// TIA Portal project "PROGRAMA_P1" (V16)

(* hardware
DEVICE "S7-1200 station_1"  S7-1200 Station
   slot 0: "Rack_0"  S7-1200 Rack  Rack  V1.0
   slot 1: "PLC_1"  CPU 1215C DC/DC/DC  6ES7 215-1AG40-0XB0  V4.4
DEVICE "PC-System_1"  SIMATIC PC station
   slot 0: "Estación PC SIMATIC"  Rail  SIMATIC PC-Station  V1.0
      slot 125: "Stationmanager"  Station_Manager  V6.0.4
   slot 1: "HMI_RT_1"  WinCC RT Advanced  6AV2 104-0xxxx-xxxx  16.0.0.0
      slot 33792: "Interfaz del equipo"  Host interface
   slot 2: "IE general_1"  IE General  IE_CP  V8.2.0
*)

// ===== PLC "PLC_1"  CPU 1215C DC/DC/DC =====

VAR_GLOBAL   // PLC tag table "Tabla de variables estándar"
   "Guardamotor 1Q1" AT %I0.0 : Bool;
   "Detector 1B1" AT %I0.1 : Bool;
   "Detector 1B2" AT %I0.2 : Bool;
   "Fotocelula 1B3" AT %I0.3 : Bool;
   "Pulsador Reinicio 1S1" AT %I0.4 : Bool;
   "Pulsador Paro 1S2" AT %I0.5 : Bool;
   "Contactor Apertura 1KM1" AT %Q0.0 : Bool;
   "Contactor Cerrado 1KM2" AT %Q0.1 : Bool;
   "Piloto 1H1" AT %Q0.2 : Bool;
   "Etapa 0" AT %M10.0 : Bool;
   "Etapa 1" AT %M10.1 : Bool;
   "Etapa 2" AT %M10.2 : Bool;
   "Etapa 3" AT %M10.3 : Bool;
   "Etapa 4" AT %M10.4 : Bool;
   "Etapa 5" AT %M10.5 : Bool;
   "Etapa 6" AT %M10.6 : Bool;
   "Etapa 7" AT %M10.7 : Bool;
   "Etapa 8" AT %M11.0 : Bool;
   "Etapa 9" AT %M11.1 : Bool;
   "Etapa 10" AT %M11.2 : Bool;
   "Etapa 11" AT %M11.3 : Bool;
   "Etapa 12" AT %M11.4 : Bool;
   "Etapa 20" AT %M11.5 : Bool;
   "Etapa 21" AT %M11.6 : Bool;
   "Etapa 22" AT %M11.7 : Bool;
   "System_Byte" AT %MB1 : Byte;
   "FirstScan" AT %M1.0 : Bool;
   "DiagStatusUpdate" AT %M1.1 : Bool;
   "AlwaysTRUE" AT %M1.2 : Bool;
   "AlwaysFALSE" AT %M1.3 : Bool;
   "Clock_Byte" AT %MB0 : Byte;
   "Clock_10Hz" AT %M0.0 : Bool;
   "Clock_5Hz" AT %M0.1 : Bool;
   "Clock_2.5Hz" AT %M0.2 : Bool;
   "Clock_2Hz" AT %M0.3 : Bool;
   "Clock_1.25Hz" AT %M0.4 : Bool;
   "Clock_1Hz" AT %M0.5 : Bool;
   "Clock_0.625Hz" AT %M0.6 : Bool;
   "Clock_0.5Hz" AT %M0.7 : Bool;
   "MB10" AT %MB10 : Byte;
   "MB11" AT %MB11 : Byte;
END_VAR

DATA_BLOCK "Variables"   // DB1
{ S7_Optimized_Access := 'TRUE' }
VERSION : 0.1
   VAR
      MAN : Bool;
      T2Time : Time;
      ActualTime : DTL;
      TimeError : Word;
      Abrir_Manual : Bool;
      Cerrar_Manual : Bool;
      InTime : Bool;
      Flanco_Paro : Bool;
      LeftTime : Time;
   END_VAR
BEGIN
END_DATA_BLOCK

// folder: System blocks/Program resources

DATA_BLOCK "T1"   // DB2
{ S7_Optimized_Access := 'TRUE' }
AUTHOR : Simatic
FAMILY : IEC
NAME : IEC_TMR
VERSION : 1.0
// stored: InstanceOfName IEC_TIMER
"IEC_TIMER"
BEGIN
END_DATA_BLOCK

DATA_BLOCK "T2"   // DB3
{ S7_Optimized_Access := 'TRUE' }
AUTHOR : Simatic
FAMILY : IEC
NAME : IEC_TMR
VERSION : 1.0
// stored: InstanceOfName IEC_TIMER
"IEC_TIMER"
BEGIN
END_DATA_BLOCK

// folder: (top level)

ORGANIZATION_BLOCK "Main"   // OB1, LAD, ProgramCycle
TITLE = "Main Program Sweep (Cycle)"
{ S7_Optimized_Access := 'TRUE' }
VERSION : 0.1
   VAR_INPUT
      Initial_Call : Bool;   // Initial call of this OB
      Remanence : Bool;   // =True, if remanent data are available
   END_VAR
BEGIN

REGION Network 1: SR Etapa 0
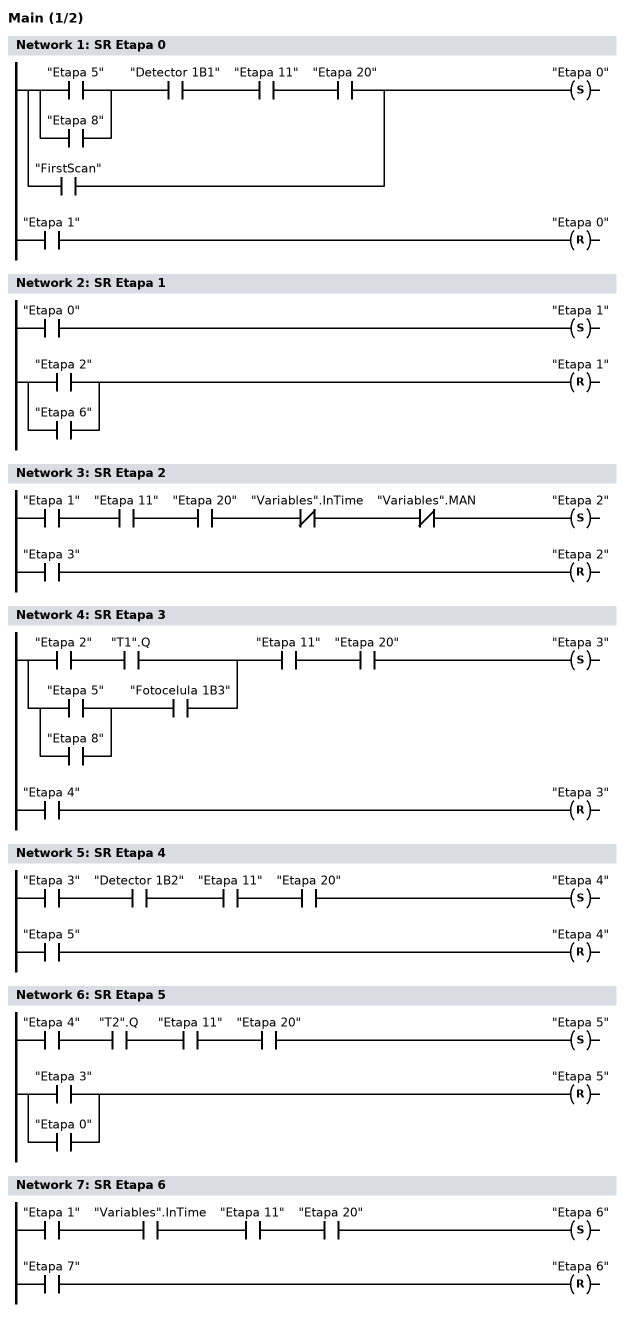
   RUNG wire#powerrail
      Contact( "Etapa 5" )
      wire#w1
      Contact( "Detector 1B1" )
      Contact( "Etapa 11" )
      Contact( "Etapa 20" )
      wire#w2
      S_Coil( "Etapa 0" )
   END_RUNG
   RUNG wire#powerrail
      Contact( "Etapa 8" )
   END_RUNG wire#w1
   RUNG wire#powerrail
      Contact( "FirstScan" )
   END_RUNG wire#w2
   RUNG wire#powerrail
      Contact( "Etapa 1" )
      R_Coil( "Etapa 0" )
   END_RUNG
   // the same network as SCL:
   IF (("Etapa 5" OR "Etapa 8") AND "Detector 1B1" AND "Etapa 11" AND "Etapa 20") OR "FirstScan" THEN
       "Etapa 0" := TRUE;
   END_IF;
   IF "Etapa 1" THEN "Etapa 0" := FALSE; END_IF;
END_REGION

REGION Network 2: SR Etapa 1
   RUNG wire#powerrail
      Contact( "Etapa 0" )
      S_Coil( "Etapa 1" )
   END_RUNG
   RUNG wire#powerrail
      Contact( "Etapa 2" )
      wire#w1
      R_Coil( "Etapa 1" )
   END_RUNG
   RUNG wire#powerrail
      Contact( "Etapa 6" )
   END_RUNG wire#w1
   // the same network as SCL:
   IF "Etapa 0" THEN "Etapa 1" := TRUE; END_IF;
   IF "Etapa 2" OR "Etapa 6" THEN "Etapa 1" := FALSE; END_IF;
END_REGION

REGION Network 3: SR Etapa 2
   RUNG wire#powerrail
      Contact( "Etapa 1" )
      Contact( "Etapa 11" )
      Contact( "Etapa 20" )
      I_Contact( "Variables".InTime )
      I_Contact( "Variables".MAN )
      S_Coil( "Etapa 2" )
   END_RUNG
   RUNG wire#powerrail
      Contact( "Etapa 3" )
      R_Coil( "Etapa 2" )
   END_RUNG
   // the same network as SCL:
   IF "Etapa 1" AND "Etapa 11" AND "Etapa 20" AND NOT "Variables".InTime AND NOT "Variables".MAN THEN
       "Etapa 2" := TRUE;
   END_IF;
   IF "Etapa 3" THEN "Etapa 2" := FALSE; END_IF;
END_REGION

REGION Network 4: SR Etapa 3
   RUNG wire#powerrail
      Contact( "Etapa 2" )
      Contact( "T1".Q )
      wire#w1
      Contact( "Etapa 11" )
      Contact( "Etapa 20" )
      S_Coil( "Etapa 3" )
   END_RUNG
   RUNG wire#powerrail
      Contact( "Etapa 5" )
      wire#w2
      Contact( "Fotocelula 1B3" )
   END_RUNG wire#w1
   RUNG wire#powerrail
      Contact( "Etapa 8" )
   END_RUNG wire#w2
   RUNG wire#powerrail
      Contact( "Etapa 4" )
      R_Coil( "Etapa 3" )
   END_RUNG
   // the same network as SCL:
   IF (("Etapa 2" AND "T1".Q) OR (("Etapa 5" OR "Etapa 8") AND "Fotocelula 1B3")) AND "Etapa 11" AND "Etapa 20" THEN
       "Etapa 3" := TRUE;
   END_IF;
   IF "Etapa 4" THEN "Etapa 3" := FALSE; END_IF;
END_REGION

REGION Network 5: SR Etapa 4
   RUNG wire#powerrail
      Contact( "Etapa 3" )
      Contact( "Detector 1B2" )
      Contact( "Etapa 11" )
      Contact( "Etapa 20" )
      S_Coil( "Etapa 4" )
   END_RUNG
   RUNG wire#powerrail
      Contact( "Etapa 5" )
      R_Coil( "Etapa 4" )
   END_RUNG
   // the same network as SCL:
   IF "Etapa 3" AND "Detector 1B2" AND "Etapa 11" AND "Etapa 20" THEN "Etapa 4" := TRUE; END_IF;
   IF "Etapa 5" THEN "Etapa 4" := FALSE; END_IF;
END_REGION

REGION Network 6: SR Etapa 5
   RUNG wire#powerrail
      Contact( "Etapa 4" )
      Contact( "T2".Q )
      Contact( "Etapa 11" )
      Contact( "Etapa 20" )
      S_Coil( "Etapa 5" )
   END_RUNG
   RUNG wire#powerrail
      Contact( "Etapa 3" )
      wire#w1
      R_Coil( "Etapa 5" )
   END_RUNG
   RUNG wire#powerrail
      Contact( "Etapa 0" )
   END_RUNG wire#w1
   // the same network as SCL:
   IF "Etapa 4" AND "T2".Q AND "Etapa 11" AND "Etapa 20" THEN "Etapa 5" := TRUE; END_IF;
   IF "Etapa 3" OR "Etapa 0" THEN "Etapa 5" := FALSE; END_IF;
END_REGION

REGION Network 7: SR Etapa 6
   RUNG wire#powerrail
      Contact( "Etapa 1" )
      Contact( "Variables".InTime )
      Contact( "Etapa 11" )
      Contact( "Etapa 20" )
      S_Coil( "Etapa 6" )
   END_RUNG
   RUNG wire#powerrail
      Contact( "Etapa 7" )
      R_Coil( "Etapa 6" )
   END_RUNG
   // the same network as SCL:
   IF "Etapa 1" AND "Variables".InTime AND "Etapa 11" AND "Etapa 20" THEN "Etapa 6" := TRUE; END_IF;
   IF "Etapa 7" THEN "Etapa 6" := FALSE; END_IF;
END_REGION

REGION Network 8: SR Etapa 7
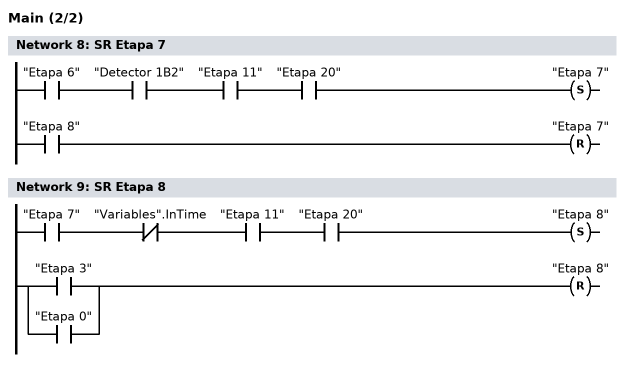
   RUNG wire#powerrail
      Contact( "Etapa 6" )
      Contact( "Detector 1B2" )
      Contact( "Etapa 11" )
      Contact( "Etapa 20" )
      S_Coil( "Etapa 7" )
   END_RUNG
   RUNG wire#powerrail
      Contact( "Etapa 8" )
      R_Coil( "Etapa 7" )
   END_RUNG
   // the same network as SCL:
   IF "Etapa 6" AND "Detector 1B2" AND "Etapa 11" AND "Etapa 20" THEN "Etapa 7" := TRUE; END_IF;
   IF "Etapa 8" THEN "Etapa 7" := FALSE; END_IF;
END_REGION

REGION Network 9: SR Etapa 8
   RUNG wire#powerrail
      Contact( "Etapa 7" )
      I_Contact( "Variables".InTime )
      Contact( "Etapa 11" )
      Contact( "Etapa 20" )
      S_Coil( "Etapa 8" )
   END_RUNG
   RUNG wire#powerrail
      Contact( "Etapa 3" )
      wire#w1
      R_Coil( "Etapa 8" )
   END_RUNG
   RUNG wire#powerrail
      Contact( "Etapa 0" )
   END_RUNG wire#w1
   // the same network as SCL:
   IF "Etapa 7" AND NOT "Variables".InTime AND "Etapa 11" AND "Etapa 20" THEN "Etapa 8" := TRUE; END_IF;
   IF "Etapa 3" OR "Etapa 0" THEN "Etapa 8" := FALSE; END_IF;
END_REGION
END_ORGANIZATION_BLOCK

ORGANIZATION_BLOCK "Temporizadores"   // OB123, LAD, ProgramCycle
TITLE = "Main Program Sweep (Cycle)"
{ S7_Optimized_Access := 'TRUE' }
VERSION : 0.1
   VAR_INPUT
      Initial_Call : Bool;   // Initial call of this OB
      Remanence : Bool;   // =True, if remanent data are available
   END_VAR
BEGIN

REGION Network 1: Temporizador 1
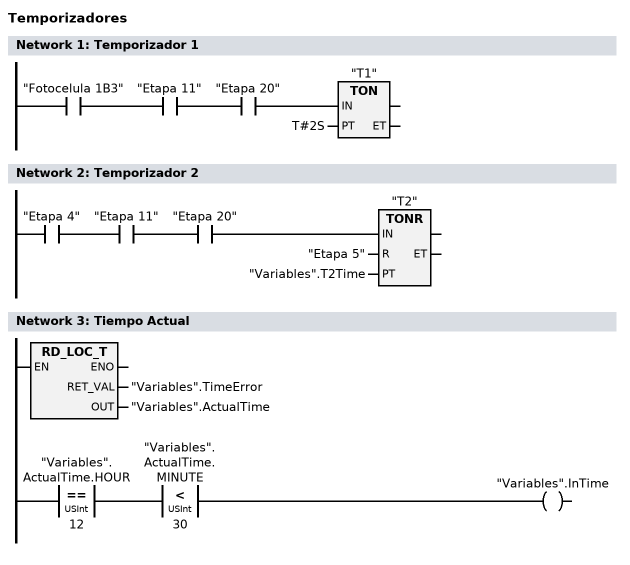
   "T1".TON(IN := "Fotocelula 1B3" AND "Etapa 11" AND "Etapa 20", PT := T#2S);
END_REGION

REGION Network 2: Temporizador 2
   "T2".TONR(IN := "Etapa 4" AND "Etapa 11" AND "Etapa 20", R := "Etapa 5", PT := "Variables".T2Time);
END_REGION

REGION Network 3: Tiempo Actual
   "Variables".TimeError := RD_LOC_T(OUT => "Variables".ActualTime);
   "Variables".InTime := ("Variables".ActualTime.HOUR = 12) AND ("Variables".ActualTime.MINUTE < 30);
END_REGION

REGION Network 4 (SCL): Cálculo tiempo restante
   "Variables".LeftTime := "T2".PT - "T2".ET;
END_REGION
END_ORGANIZATION_BLOCK

ORGANIZATION_BLOCK "Tratamiento Posterior"   // OB124, LAD, ProgramCycle
TITLE = "Main Program Sweep (Cycle)"
{ S7_Optimized_Access := 'TRUE' }
VERSION : 0.1
   VAR_INPUT
      Initial_Call : Bool;   // Initial call of this OB
      Remanence : Bool;   // =True, if remanent data are available
   END_VAR
BEGIN

REGION Network 1: 1KM1
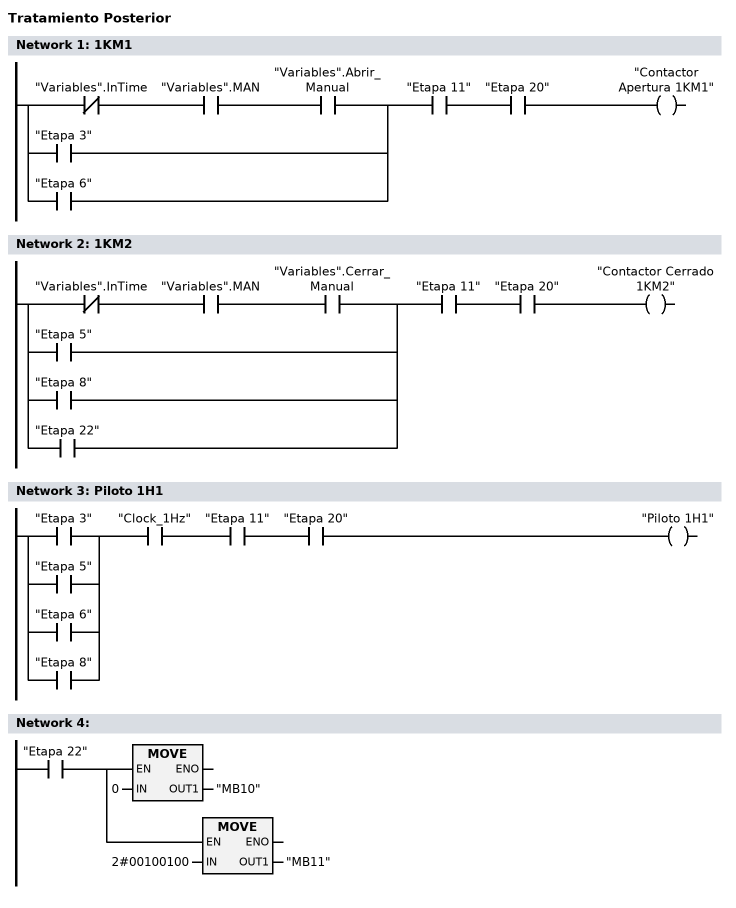
   RUNG wire#powerrail
      I_Contact( "Variables".InTime )
      Contact( "Variables".MAN )
      Contact( "Variables".Abrir_Manual )
      wire#w1
      Contact( "Etapa 11" )
      Contact( "Etapa 20" )
      Coil( "Contactor Apertura 1KM1" )
   END_RUNG
   RUNG wire#powerrail
      Contact( "Etapa 3" )
   END_RUNG wire#w1
   RUNG wire#powerrail
      Contact( "Etapa 6" )
   END_RUNG wire#w1
   // the same network as SCL:
   "Contactor Apertura 1KM1" := ((NOT "Variables".InTime AND "Variables".MAN AND "Variables".Abrir_Manual) OR "Etapa 3" OR "Etapa 6") AND "Etapa 11" AND "Etapa 20";
END_REGION

REGION Network 2: 1KM2
   RUNG wire#powerrail
      I_Contact( "Variables".InTime )
      Contact( "Variables".MAN )
      Contact( "Variables".Cerrar_Manual )
      wire#w1
      Contact( "Etapa 11" )
      Contact( "Etapa 20" )
      Coil( "Contactor Cerrado 1KM2" )
   END_RUNG
   RUNG wire#powerrail
      Contact( "Etapa 5" )
   END_RUNG wire#w1
   RUNG wire#powerrail
      Contact( "Etapa 8" )
   END_RUNG wire#w1
   RUNG wire#powerrail
      Contact( "Etapa 22" )
   END_RUNG wire#w1
   // the same network as SCL:
   "Contactor Cerrado 1KM2" := ((NOT "Variables".InTime AND "Variables".MAN AND "Variables".Cerrar_Manual) OR "Etapa 5" OR "Etapa 8" OR "Etapa 22") AND "Etapa 11" AND "Etapa 20";
END_REGION

REGION Network 3: Piloto 1H1
   RUNG wire#powerrail
      Contact( "Etapa 3" )
      wire#w1
      Contact( "Clock_1Hz" )
      Contact( "Etapa 11" )
      Contact( "Etapa 20" )
      Coil( "Piloto 1H1" )
   END_RUNG
   RUNG wire#powerrail
      Contact( "Etapa 5" )
   END_RUNG wire#w1
   RUNG wire#powerrail
      Contact( "Etapa 6" )
   END_RUNG wire#w1
   RUNG wire#powerrail
      Contact( "Etapa 8" )
   END_RUNG wire#w1
   // the same network as SCL:
   "Piloto 1H1" := ("Etapa 3" OR "Etapa 5" OR "Etapa 6" OR "Etapa 8") AND "Clock_1Hz" AND "Etapa 11" AND "Etapa 20";
END_REGION

REGION Network 4
   RUNG wire#powerrail
      Contact( "Etapa 22" )
      wire#w1
      Move(in := 0, out1 => "MB10")
   END_RUNG
   RUNG wire#w1
      Move(in := 2#00100100, out1 => "MB11")
   END_RUNG
   // the same network as SCL:
   IF "Etapa 22" THEN
       "MB10" := 0;
       "MB11" := 2#00100100;
   END_IF;
END_REGION
END_ORGANIZATION_BLOCK

ORGANIZATION_BLOCK "Paro"   // OB125, LAD, ProgramCycle
TITLE = "Main Program Sweep (Cycle)"
{ S7_Optimized_Access := 'TRUE' }
VERSION : 0.1
   VAR_INPUT
      Initial_Call : Bool;   // Initial call of this OB
      Remanence : Bool;   // =True, if remanent data are available
   END_VAR
   VAR_TEMP   // added for the SCL form of the ladder/FBD networks
      _w1 : Bool;
   END_VAR
BEGIN

REGION Network 1: SR Etapa 20
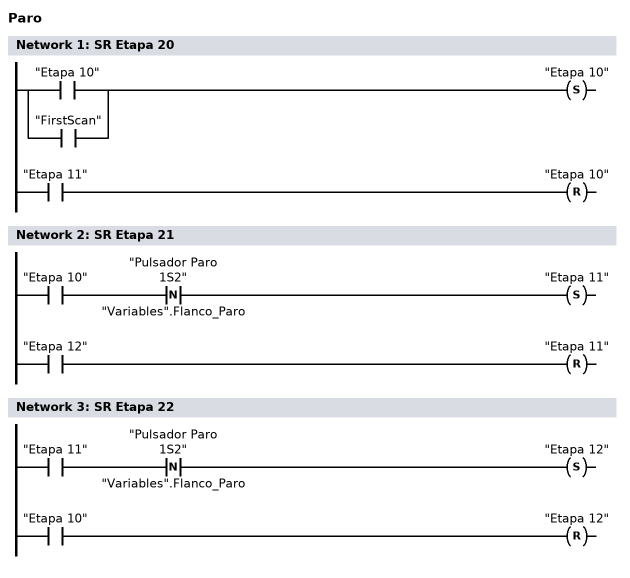
   RUNG wire#powerrail
      Contact( "Etapa 10" )
      wire#w1
      S_Coil( "Etapa 10" )
   END_RUNG
   RUNG wire#powerrail
      Contact( "FirstScan" )
   END_RUNG wire#w1
   RUNG wire#powerrail
      Contact( "Etapa 11" )
      R_Coil( "Etapa 10" )
   END_RUNG
   // the same network as SCL:
   IF "Etapa 10" OR "FirstScan" THEN "Etapa 10" := TRUE; END_IF;
   IF "Etapa 11" THEN "Etapa 10" := FALSE; END_IF;
END_REGION

REGION Network 2: SR Etapa 21
   RUNG wire#powerrail
      Contact( "Etapa 10" )
      N_Contact(operand := "Pulsador Paro 1S2", bit := "Variables".Flanco_Paro)
      S_Coil( "Etapa 11" )
   END_RUNG
   RUNG wire#powerrail
      Contact( "Etapa 12" )
      R_Coil( "Etapa 11" )
   END_RUNG
   // the same network as SCL:
   #_w1 := "Etapa 10" AND NOT "Pulsador Paro 1S2" AND "Variables".Flanco_Paro;   // falling edge of "Pulsador Paro 1S2"
   "Variables".Flanco_Paro := "Pulsador Paro 1S2";
   IF #_w1 THEN "Etapa 11" := TRUE; END_IF;
   IF "Etapa 12" THEN "Etapa 11" := FALSE; END_IF;
END_REGION

REGION Network 3: SR Etapa 22
   RUNG wire#powerrail
      Contact( "Etapa 11" )
      N_Contact(operand := "Pulsador Paro 1S2", bit := "Variables".Flanco_Paro)
      S_Coil( "Etapa 12" )
   END_RUNG
   RUNG wire#powerrail
      Contact( "Etapa 10" )
      R_Coil( "Etapa 12" )
   END_RUNG
   // the same network as SCL:
   #_w1 := "Etapa 11" AND NOT "Pulsador Paro 1S2" AND "Variables".Flanco_Paro;   // falling edge of "Pulsador Paro 1S2"
   "Variables".Flanco_Paro := "Pulsador Paro 1S2";
   IF #_w1 THEN "Etapa 12" := TRUE; END_IF;
   IF "Etapa 10" THEN "Etapa 12" := FALSE; END_IF;
END_REGION
END_ORGANIZATION_BLOCK

ORGANIZATION_BLOCK "Reset"   // OB126, LAD, ProgramCycle
TITLE = "Main Program Sweep (Cycle)"
{ S7_Optimized_Access := 'TRUE' }
VERSION : 0.1
   VAR_INPUT
      Initial_Call : Bool;   // Initial call of this OB
      Remanence : Bool;   // =True, if remanent data are available
   END_VAR
BEGIN

REGION Network 1: SR Etapa 20
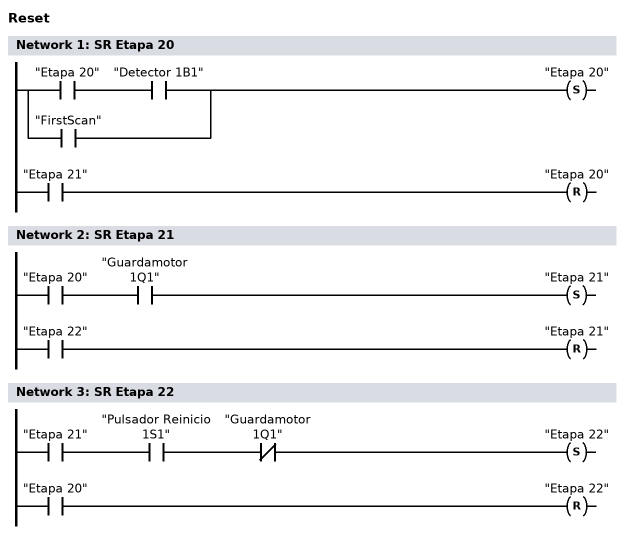
   RUNG wire#powerrail
      Contact( "Etapa 20" )
      Contact( "Detector 1B1" )
      wire#w1
      S_Coil( "Etapa 20" )
   END_RUNG
   RUNG wire#powerrail
      Contact( "FirstScan" )
   END_RUNG wire#w1
   RUNG wire#powerrail
      Contact( "Etapa 21" )
      R_Coil( "Etapa 20" )
   END_RUNG
   // the same network as SCL:
   IF ("Etapa 20" AND "Detector 1B1") OR "FirstScan" THEN "Etapa 20" := TRUE; END_IF;
   IF "Etapa 21" THEN "Etapa 20" := FALSE; END_IF;
END_REGION

REGION Network 2: SR Etapa 21
   RUNG wire#powerrail
      Contact( "Etapa 20" )
      Contact( "Guardamotor 1Q1" )
      S_Coil( "Etapa 21" )
   END_RUNG
   RUNG wire#powerrail
      Contact( "Etapa 22" )
      R_Coil( "Etapa 21" )
   END_RUNG
   // the same network as SCL:
   IF "Etapa 20" AND "Guardamotor 1Q1" THEN "Etapa 21" := TRUE; END_IF;
   IF "Etapa 22" THEN "Etapa 21" := FALSE; END_IF;
END_REGION

REGION Network 3: SR Etapa 22
   RUNG wire#powerrail
      Contact( "Etapa 21" )
      Contact( "Pulsador Reinicio 1S1" )
      I_Contact( "Guardamotor 1Q1" )
      S_Coil( "Etapa 22" )
   END_RUNG
   RUNG wire#powerrail
      Contact( "Etapa 20" )
      R_Coil( "Etapa 22" )
   END_RUNG
   // the same network as SCL:
   IF "Etapa 21" AND "Pulsador Reinicio 1S1" AND NOT "Guardamotor 1Q1" THEN "Etapa 22" := TRUE; END_IF;
   IF "Etapa 20" THEN "Etapa 22" := FALSE; END_IF;
END_REGION
END_ORGANIZATION_BLOCK

(* ===== HMI "HMI_RT_1" =====
system functions are stored by id; their names below are inferred from use
connection "HMI_Conexión_1": ETHERNET, S7_1200_OMS

HMI tags "Tabla de variables estándar"
   "Variables_T2Time" : Time = PLC Variables.T2Time, 1 s
   "Variables_MAN" : Bool = PLC Variables.MAN, 1 s
   "Variables_Abrir_Manual" : Bool = PLC Variables.Abrir_Manual, 1 s
   "Variables_Cerrar_Manual" : Bool = PLC Variables.Cerrar_Manual, 1 s
   "Variables_LeftTime" : Time = PLC Variables.LeftTime, 1 s

screen "Imagen_1" 800x600
   IOField "Campo ES_1" at 280,177 size 66x37; FormatPattern 99999
      ProcessValue <- "Variables_T2Time"
   TextField "Campo de texto_1" at 265,65 size 269x22; Text 'Tiempo de apertura de puerta (ms):'
   Switch "Interruptor_1" at 330,302 size 129x60; CaptionText 'Switch'; TextOff 'AUTO'; TextOn 'MAN'
      ProcessValue <- "Variables_MAN"
   Button "Botón_1" at 347,408 size 96x32; TextOff 'Abrir'
      on Press: SetBit("Variables_Abrir_Manual")
      on Release: ResetBit("Variables_Abrir_Manual")
   Button "Botón_2" at 347,491 size 96x32; TextOff 'Cerrar'
      on Press: SetBit("Variables_Cerrar_Manual")
      on Release: ResetBit("Variables_Cerrar_Manual")
   Gauge "Indicador gauge_1" at 394,130 size 140x140; CaptionText 'SIMATIC'; UnitText 'Unit'
      MaximumValue <- "Variables_T2Time"
      ProcessValue <- "Variables_LeftTime"
*)